// Implicitly generated code : DO NOT EDIT
FUNCTION CheckLRangeSigned : LINT
VAR_INPUT
	value, lower, upper: LINT;
END_VAR

// Implicitly generated code : Only an Implementation suggestion
{noflow}
Fault_Count_G(CU:=FALSE) ; 
IF (value < lower) THEN
	CheckLRangeSigned := lower;
		Fault_Count_G(CU:=TRUE) ; 
ELSIF(value > upper) THEN
	CheckLRangeSigned := upper;
		Fault_Count_G(CU:=TRUE) ; 
ELSE
	CheckLRangeSigned := value;
END_IF

{flow}

END_FUNCTION

(* stored: Version 1.1.0.1, ProductVersion 3.1.4024.2
   POU CheckLRangeSigned: Id {cffc36fe-83b5-4c00-b686-90a3b745eec4}, SpecialFunc CheckLRangeSigned *)
